{attribute 'qualified_only'}
VAR_GLOBAL
	
	{attribute 'OPC.UA.DA' := '1'} OPC_TemperatureContactor : BOOL; // Temperature contactor
	{attribute 'OPC.UA.DA' := '1'} OPC_ReactorTemperature : INT; // Reactor temperature
	{attribute 'OPC.UA.DA' := '1'} OPC_ReactorLowerTemperature : INT; // Reactor temperature
	{attribute 'OPC.UA.DA' := '1'} OPC_ReactorPressure : INT; // Reactor pressure
	{attribute 'OPC.UA.DA' := '1'} OPC_ReactorTemperatureSetpoint: INT; // Reactr temperature setpoint
	{attribute 'OPC.UA.DA' := '1'} OPC_SlurryInletValve: BOOL;
	{attribute 'OPC.UA.DA' := '1'} OPC_SlurryOutletValve: BOOL;
	{attribute 'OPC.UA.DA' := '1'} OPC_ExtractiveOutletOnOffValve: BOOL;
	{attribute 'OPC.UA.DA' := '1'} OPC_ExtractiveControlValveOpening: INT;
	
	{attribute 'OPC.UA.DA' := '1'} OPC_PumpingPressure: DINT;
	{attribute 'OPC.UA.DA' := '1'} OPC_PumpingPressureSetpoint: DINT;
	
	{attribute 'OPC.UA.DA' := '1'} OPC_PreHeaterTemperature: DINT;
	{attribute 'OPC.UA.DA' := '1'} OPC_PreHeaterTemperatureSetpoint: DINT;
	
	{attribute 'OPC.UA.DA' := '1'} OPC_SeparatorTemperature: DINT;
	{attribute 'OPC.UA.DA' := '1'} OPC_SeparatorTemperatureSetpoint: DINT;
	
	{attribute 'OPC.UA.DA' := '1'} OPC_CO2VolumetricFlow: REAL;
	
	{attribute 'OPC.UA.DA' := '1'} OPC_AutoExtractionState: STRING;
	
	// Program name 
	{attribute 'OPC.UA.DA' := '1'} OPC_ProgramNamePrefix: STRING;
	
	// Special data 
	{attribute 'OPC.UA.DA' := '1'} OPC_OutletValveOpenArray: ARRAY[0..99] OF BOOL;
	{attribute 'OPC.UA.DA' := '1'} OPC_OutletValveOpenTimeStampArray: ARRAY[0..99] OF DT;
	{attribute 'OPC.UA.DA' := '1'} OPC_OutletValveCloseArray: ARRAY[0..99] OF BOOL;
	{attribute 'OPC.UA.DA' := '1'} OPC_OutletValveCloseTimeStampArray: ARRAY[0..99] OF DT;
END_VAR

(* stored: Version 1.1.0.1, ProductVersion 3.1.4024.9
   GVL GVL_OPC: Id {ff69d8bd-4aa9-4fbf-a8cd-ee3ab3220a99} *)
